// SIMATIC STEP 7 (V5.x) project Skipenes
// CPU: CPU315-2 DP(1)

SYMBOL_TABLE
"Obstruction"	I 8.0	BOOL	// [input]
"Stop button"	I 8.1	BOOL	// [input]
"Cab order 1 button"	I 8.2	BOOL	// [input] Goto floor 1
"Cab order 2 button"	I 8.3	BOOL	// [input] Goto floor 2
"Cab order 3 button"	I 8.4	BOOL	// [input] Goto floor 3
"Cab order 4 button"	I 8.5	BOOL	// [input] Goto floor 4
"Up 1 button"	I 8.6	BOOL	// [input] 1st floor. direction up
"Up 2 button"	I 8.7	BOOL	// [input] 2nd floor. direction up
"Down 2 button"	I 9.0	BOOL	// [input] 2nd floor. direction down
"Up 3 button"	I 9.1	BOOL	// [input] 3rd floor. direction up
"Down 3 button"	I 9.2	BOOL	// [input] 3rd floor. direction down
"Down 4 button"	I 9.3	BOOL	// [input] 4th floor. direction down
"Floor sensor 1"	I 9.4	BOOL	// [input]
"Floor sensor 2"	I 9.5	BOOL	// [input]
"Floor sensor 3"	I 9.6	BOOL	// [input]
"Floor sensor 4"	I 9.7	BOOL	// [input]
"main"	OB 1	OB 1
"Motor drive strength"	PQW 272	WORD
"Motor direction"	Q 8.0	BOOL	// 0 = up, 1 = down
"Stop button light"	Q 8.1	BOOL	// [output]
"Cab order 1 light"	Q 8.2	BOOL	// [output] floor 1 queued
"Cab order 2 light"	Q 8.3	BOOL	// [output] floor 2 queued
"Cab order 3 light"	Q 8.4	BOOL	// [output] floor 3 queued
"Cab order 4 light"	Q 8.5	BOOL	// [output] floor 4 queued
"Up 1 light"	Q 8.6	BOOL	// [output] 1st floor. direction up
"Up 2 light"	Q 8.7	BOOL	// [output] 2nd floor. direction up
"Down 2 light"	Q 9.0	BOOL	// [output] 2nd floor. direction down
"Up 3 light"	Q 9.1	BOOL	// [output] 3rd floor. direction up
"Down 3 light"	Q 9.2	BOOL	// [output] 3rd floor. direction down
"Down 4 light"	Q 9.3	BOOL	// [output] 4th floor. direction down
"Door open"	Q 9.4	BOOL	// [output] light indicating open door
"unused"	Q 9.5	BOOL
"Floor indicator bit 1"	Q 9.6	BOOL	// on for 2nd and 4th floor
"Floor indicator bit 2"	Q 9.7	BOOL	// on for 3rd and 4th floor
END_SYMBOL_TABLE
